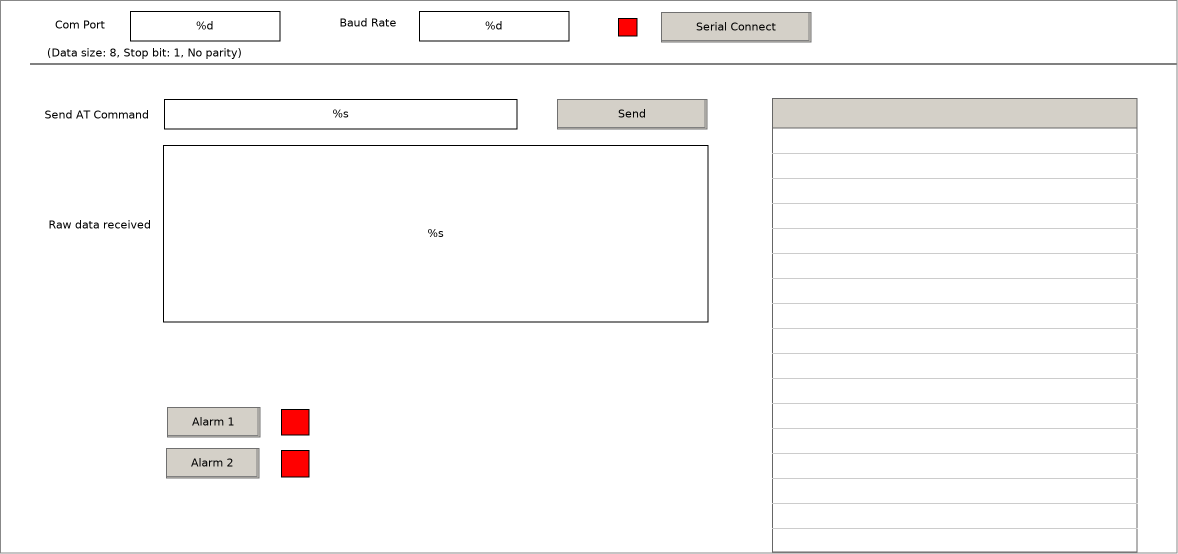
VISUALIZATION Visualization  // 1178x554
    Button (661,12 150x30), "Serial Connect"
        toggle MAIN.bSerial
    Rectangle (130,11 150x30), "%d", text variable: MAIN.stSerialCfg.ComPort
        OnMouseDown: write the text variable via Default
    Rectangle (419,11 150x30), "%d", text variable: MAIN.stSerialCfg.Baudrate
        OnMouseDown: write the text variable via Default
    Label (5,10 150x30), "Com Port"
    Label (293,8 150x30), "Baud Rate"
    Rectangle (164,99 353x30), "%s", text variable: MAIN.sATCommand
        OnMouseDown: write the text variable via Default
    Label (22,100 150x30), "Send AT Command"
    Label (25,210 150x30), "Raw data received"
    Rectangle (163,145 545x177), "%s", text variable: MAIN.sRawReceive
    Button (557,99 150x30), "Send"
        toggle MAIN.bSend
    Rectangle (618,18 19x18), colour toggle: MAIN.bPortOpened
    Rectangle (281,409 28x26), colour toggle: MAIN.alarm
    Rectangle (281,450 28x27), colour toggle: MAIN.alarm2
    Button (167,407 93x30), "Alarm 1"
        toggle MAIN.alarm
    Button (166,448 93x30), "Alarm 2"
        toggle MAIN.alarm2
    Table (772,98 365x454), data array: MAIN.arrStr
        p3854506369: MAIN.arrStr[INDEX]
        p2232123230: Received SMS
    Line (1176,64) (30,64)
    Label (15,38 259x30), "(Data size: 8, Stop bit: 1, No parity)"
END_VISUALIZATION

(* stored: Version 1.1.0.1, ProductVersion 3.1.4020.6
   Visu Visualization: Id {245ddf28-826a-4683-8ab3-dfd4d2347a35} *)
